{attribute addProperty BoxType "EPP1518-0002-0016"}
{attribute addProperty Id "StatusAT %I*Status_CCE4E0C81620Counter_valueAT %I*UDINT32417"}
{attribute addProperty CRC "1239498684"}
{attribute addProperty SizeInBites "48"}
{attribute addProperty SizeInBytes "6"}
TYPE CNT_Input_Channel_49E13FBC :
STRUCT
	{attribute addProperty Name "Status"}
	Status AT %I* : Status_CCE4E0C8;
	{attribute addProperty Name "Counter_value"}
	Counter_value AT %I* : UDINT;
END_STRUCT
END_TYPE

(* stored: Version 1.2.0.0, ProductVersion 3.1.4024.9
   DUT CNT_Input_Channel_49E13FBC: Id {2b6ca3a7-3cc0-429b-adc6-86360ee998df} *)
